{attribute addProperty BoxType "AT2050-0501-0019"}
{attribute addProperty Id "A_0081_AT2002_5250_0018_AT2002_5250AT2002_C5E5984862678.25"}
{attribute addProperty CRC "219124159"}
{attribute addProperty SizeInBites "626"}
{attribute addProperty SizeInBytes "78.25"}
TYPE A_0069_AT2050_0501_0019_AT2050_0501_0D0F91BF EXTENDS AT2050_BA5A9548 :
STRUCT
	{attribute addProperty Name "A_0081_AT2002_5250_0018_AT2002_5250"}
	A_0081_AT2002_5250_0018_AT2002_5250 : AT2002_C5E59848;
END_STRUCT
END_TYPE

(* stored: Version 1.2.0.0, ProductVersion 3.1.4024.9
   DUT A_0069_AT2050_0501_0019_AT2050_0501_0D0F91BF: Id {3ae4ed10-0fa6-4301-8841-4c89e6eff7d3} *)
